FUNCTION_BLOCK FB_Convert_2Windspeed
VAR_INPUT
	iInput			:	INT;
	tRefresh		:	TIME;
END_VAR
VAR_OUTPUT
	wOutMS			:	WORD;
	wOutKMH			:	WORD;
END_VAR
VAR
	rX				:	REAL;
	tonBlock		:	TON;
END_VAR

// For Convertion of 0-10V Signal from 0-100%
tonBlock(IN := NOT tonBlock.Q, PT := tRefresh);

IF tonBlock.Q THEN

	rX := iInput / 936.2; //Annahme 35m/s entspr. 32767
	wOutMS := REAL_TO_WORD(rX * 10);
	
	wOutKMH := REAL_TO_WORD((rX * 3.6) * 10);
	
END_IF

END_FUNCTION_BLOCK

(* stored: Version 1.1.0.1, ProductVersion 3.1.4024.13
   POU FB_Convert_2Windspeed: Id {c70ca251-9ed5-4c1b-a2b7-49705b1fa988}, SpecialFunc None *)
